# EPICS autosave request: support/calc-2-8/calcApp/Db/FuncGen_settings.req
$(P)$(Q):Amplitude
$(P)$(Q):Offset
$(P)$(Q):Frequency
$(P)$(Q):Period
$(P)$(Q):OutDrive.OUT
#$(P)$(Q):EnableOutput
#$(P)$(Q):Tran.SCAN
$(P)$(Q):Output.DRVH
$(P)$(Q):Output.DRVL
$(P)$(Q):Function
$(P)$(Q):ChartPeriod
